// TIA Portal V16 export
// export: Created 2021-07-12T14:47:18.4920294Z, ExportSetting WithDefaults, DisplayName Totally Integrated Automation Portal, DisplayVersion V16, DisplayName TIA Portal Version Control Interface, DisplayVersion V16, DisplayName TIA Portal Openness, DisplayVersion V16, DisplayName STEP 7 Professional, DisplayVersion V16, DisplayName STEP 7 Safety, DisplayVersion V16, DisplayName WinCC Professional, DisplayVersion V16
TYPE "SimaHydTO_typeHMIConnectionBasicAxislStatusDirectOutput"
TITLE = SimaHydTO_typeHMIConnectionBasicAxislStatusDirectOutput
// Direct output status
// stored: IsFailsafeCompliant false
   STRUCT
      active : Bool;   // displays activity of direct output operation
      rampingDown : Bool;   // ramping down due to positioning limits
      minSafetyPositionOverrun : Bool;   // the min. safety position was passed
      maxSafetyPositionOverrun : Bool;   // the max. safety position was passed
   END_STRUCT;
END_TYPE
